GLOBALCONSTANTS DefaultPool (* Global constants *)
  PACKAGE test::FBs::Baumsetzer::Constants;
  VAR_GLOBAL CONSTANT
    ISO_DESIGNATOR_WIDTH : UINT := 80;
    ISO_DESIGNATOR_HEIGHT : UINT := 80;
    ISO_MASK_SIZE : UINT := 480;
    ISO_VERSION_LABEL : STRING;
    MASK_WIDTH : UINT := 480;
    MASK_HEIGHT : UINT := 480;
    WorkingSet : UINT := 0;
    Macro_Reset_Einsatzdauer : UINT := 1;
    Macro_Reset_Baeume_gepflanzt : UINT := 2;
    Macro_Go_To_DataMask_Abstaende : UINT := 3;
    Macro_Go_To_DataMask_Main : UINT := 4;
    Macro_Go_To_DataMask_Manuell : UINT := 5;
    Macro_Go_To_DataMask_Geschwindigkeitssignal : UINT := 6;
    DataMask_Main : UINT := 1000;
    DataMask_Einstellungen : UINT := 1001;
    DataMask_Manuel : UINT := 1002;
    DataMask_Geschwindigkeitssignale : UINT := 1003;
    SoftKeyMask_S1 : UINT := 4000;
    Start : UINT := 5000;
    Stop : UINT := 5001;
    SoftKey_Scheinwerfer : UINT := 5002;
    SoftKey_Manuell : UINT := 5003;
    SoftKey_Einstellungen : UINT := 5004;
    SoftKey_Geschwindigkeiten : UINT := 5005;
    Button_Granulatschieber : UINT := 6000;
    Button_Reset_Einsatzdauer : UINT := 6001;
    Button_Summer : UINT := 6002;
    Button_Luftventil : UINT := 6003;
    Button_Wasserpumpe : UINT := 6004;
    Button_Wasserventil : UINT := 6005;
    Button_WBSD : UINT := 6006;
    Button_VDS : UINT := 6007;
    Button_GBSD : UINT := 6008;
    Button_MSS : UINT := 6009;
    Button_Zurueck : UINT := 6010;
    Button_Reset_Baeume_gepflanzt : UINT := 6011;
    Button_NMEA : UINT := 6012;
    InputNumber_Pflanzabstand : UINT := 9001;
    InputNumber_Luftversatz : UINT := 9002;
    InputNumber_Wasserversatz : UINT := 9003;
    InputNumber_Granulatversatz : UINT := 9004;
    InputNumber_Summer_Dauer : UINT := 9005;
    InputNumber_Luft_Dauer : UINT := 9006;
    InputNumber_Wasser_Dauer : UINT := 9007;
    InputNumber_Granulat_Dauer : UINT := 9008;
    OutputString_11000 : UINT := 11000;
    OutputString_cm : UINT := 11005;
    OutputString_Einstellungen_1 : UINT := 11006;
    OutputString_11007 : UINT := 11007;
    OutputString_11008 : UINT := 11008;
    OutputString_11009 : UINT := 11009;
    OutputString_11010 : UINT := 11010;
    OutputString_11011 : UINT := 11011;
    OutputString_11012 : UINT := 11012;
    OutputString_11013 : UINT := 11013;
    OutputString_11014 : UINT := 11014;
    OutputString_11015 : UINT := 11015;
    OutputString_11016 : UINT := 11016;
    OutputString_11017 : UINT := 11017;
    OutputString_11018 : UINT := 11018;
    OutputString_11019 : UINT := 11019;
    OutputString_11020 : UINT := 11020;
    OutputString_11021 : UINT := 11021;
    OutputString_m : UINT := 11022;
    OutputString_11023 : UINT := 11023;
    OutputString_11024 : UINT := 11024;
    OutputString_11025 : UINT := 11025;
    OutputString_11026 : UINT := 11026;
    OutputString_11027 : UINT := 11027;
    OutputString_11028 : UINT := 11028;
    OutputString_11029 : UINT := 11029;
    OutputString_11031 : UINT := 11031;
    OutputString_11032 : UINT := 11032;
    OutputString_11033 : UINT := 11033;
    OutputString_11036 : UINT := 11036;
    OutputString_11004 : UINT := 11050;
    OutputNumber_12000 : UINT := 12000;
    Einsatzstunden : UINT := 12001;
    Einsatzminuten : UINT := 12002;
    OutputNumber_Baeume_gepflanzt : UINT := 12003;
    OutputNumber_12004 : UINT := 12004;
    OutputNumber_12005 : UINT := 12005;
    OutputNumber_12006 : UINT := 12006;
    OutputNumber_12007 : UINT := 12007;
    Maschine_small : UINT := 20000;
    logo_grafinger_small : UINT := 20001;
    headlight_small : UINT := 20002;
    Zurueck_small : UINT := 20033;
    Einstellungen_small : UINT := 20501;
    pause_s : UINT := 20502;
    Manueller_Modus_small : UINT := 20503;
    gps_wheel_speed_small : UINT := 20504;
    Start_small : UINT := 20535;
    NumberVariable_Baumzaehler : UINT := 21000;
    NumberVariable_Einsatzdauer_Minuten : UINT := 21001;
    NumberVariable_Einsatzdauer_Stunden : UINT := 21002;
    FontAttributes_6x8 : UINT := 23000;
    FontAttributes_12x16 : UINT := 23001;
    FontAttributes_16x24 : UINT := 23004;
    ObjectPointer_NULL : UINT := 27000;
  END_VAR
END_GLOBALCONSTANTS
